{attribute 'enable_dynamic_creation'}
FUNCTION_BLOCK FB_Square IMPLEMENTS I_Shape
VAR_INPUT
END_VAR
VAR_OUTPUT
END_VAR
VAR
END_VAR

{warning 'Agregar implementación de método'}
METHOD M_Draw : BOOL
ADSLOGSTR(ADSLOG_MSGTYPE_HINT, 'Square', '');
M_Draw := TRUE;
END_METHOD

END_FUNCTION_BLOCK

(* stored: Version 1.1.0.1, ProductVersion 3.1.4024.12
   POU FB_Square: Id {23435c1e-9e24-49e2-a19f-fbbf3c4adf36}, SpecialFunc None
   Method M_Draw: Id {c62d25ec-9308-461b-98be-565313cc7da3} *)
